// TIA Portal V21 export
// export: Created 2026-09-06T18:39:47.503293Z, ExportSetting WithDefaults, DisplayName Totally Integrated Automation Portal, DisplayVersion V21 Hotfix 1, DisplayName STEP 7 Professional, DisplayVersion V21, DisplayName STEP 7 CFC, DisplayVersion V21, DisplayName STEP 7 Safety, DisplayVersion V21, DisplayName Tech WebApplication, DisplayVersion V21, DisplayName WinCC Basic/Comfort/Advanced, DisplayVersion V21, DisplayName SIMATIC Visualization Architect, DisplayVersion V21, DisplayName WinCC Unified, DisplayVersion V21, DisplayName SIMATIC Visualization Architect, DisplayVersion V21
VAR_GLOBAL   // PLC tag table "Marcadores_Internos"
   OK_SISTEMA AT %M0.0 : Bool;   // Permissivo geral do sistema (calculado em FC1)
   AUT_LINHA_LIGADA AT %M0.1 : Bool;   // Selo da linha em modo automatico (FC3)
   MODO_MANUAL AT %M0.2 : Bool;   // Modo manual selecionado (FC2)
   CICLO_RECUO AT %M0.3 : Bool;   // Ciclo de recuo do cilindro hidraulico (FC4)
   EMERGENCIA AT %M0.4 : Bool;   // Paragem de emergencia ativa (FC1)
   ETAPA_GRAFCET AT %MW2 : Word;   // Variavel de etapa atual do GRAFCET (FC5_GRAFCET)
   INATIVIDADE_ATIVA AT %M0.5 : Bool;   // Timer de inatividade ativo; linha sem material durante 30 s
END_VAR
